// TIA Portal V21 export
// export: Created 2000-01-01T00:00:00.0000000Z, ExportSetting None
VAR_GLOBAL   // PLC tag table "MCP_E2E"
   StartPB AT %I0.0 : Bool;
   StopPB AT %I0.1 : Bool;
   EStop AT %I0.2 : Bool;
   RunOut AT %Q0.0 : Bool;
END_VAR
